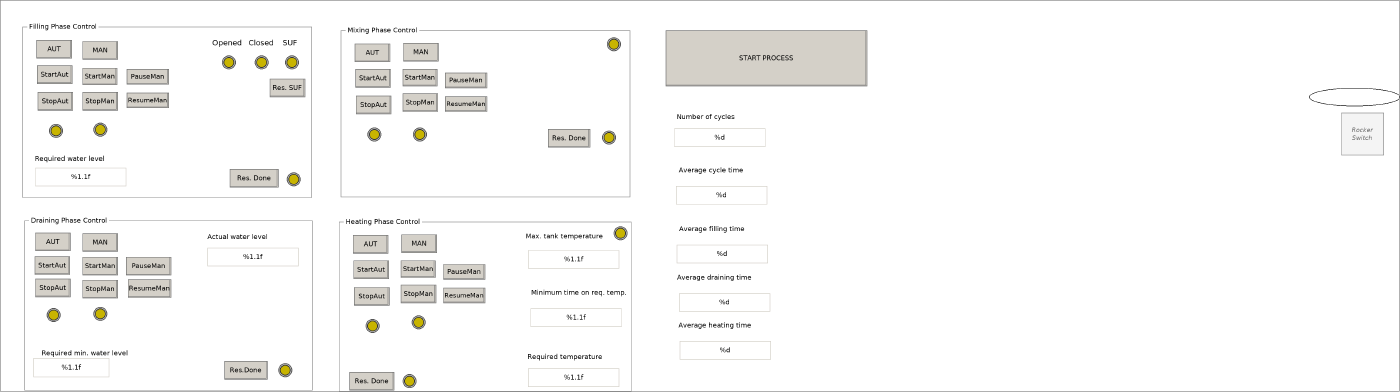
VISUALIZATION Visualization  // 2309x647
    GroupBox (40,356 475x288), "Draining Phase Control"
        Button (18,28 58x30), "AUT"
            OnMouseClick: toggle Global.Tank1.Draining.Cmd.AutCtrl
        Button (96,29 58x30), "MAN"
            OnMouseClick: toggle Global.Tank1.Draining.Cmd.ManCtrl
        Button (17,67 58x30), "StartAut"
            OnMouseClick: toggle Global.Tank1.Draining.Cmd.StartAut
        Button (168,68 74x30), "PauseMan"
            OnMouseClick: toggle Global.Tank1.Draining.Cmd.PauseMan
        Button (96,68 58x30), "StartMan"
            OnMouseClick: toggle Global.Tank1.Draining.Cmd.StartMan
        Button (96,106 58x30), "StopMan"
            OnMouseClick: toggle Global.Tank1.Draining.Cmd.StopMan
        Button (171,105 71x30), "ResumeMan"
            OnMouseClick: toggle Global.Tank1.Draining.Cmd.ResumeMan
        Button (18,104 58x30), "StopAut"
            OnMouseClick: toggle Global.Tank1.Draining.Cmd.StopAut
        Button (330,240 71x30), "Res.Done"
            OnMouseClick: toggle Global.Tank1.Draining.Cmd.ResetDone
        Lamp1 (417,242 27x26), variable: Global.Tank1.Draining.State.Done, style: Lamp-Lamp1-Yellow
        Lamp1 (35,151 27x26), variable: Global.Tank1.Draining.State.AutCtrl, style: Lamp-Lamp1-Yellow
        Lamp1 (112,149 27x26), variable: Global.Tank1.Draining.State.ManCtrl, style: Lamp-Lamp1-Yellow
        Textfield (302,53 150x30), "%1.1f", text variable: Global.Tank1.Draining.WaterLevel
        Textfield (15,235 125x31), "%1.1f", text variable: Global.Tank1.Draining.ParamDrainLevel
            OnMouseDown: write Global.Tank1.Draining.ParamDrainLevel via Edit
        Label (277,20 150x30), "Actual water level"
        Label (25,212 150x30), "Required min. water level"
    RockerSwitch (2212,186 70x70), behaviour: TOGGLE, style: Switch-RockerSwitch-Gray
    Ellipse (2159,145 150x30)
    GroupBox (37,36 477x290), "Filling Phase Control"
        Button (23,30 58x30), "AUT", text variable: Global.Tank1.Filling.Cmd.AutCtrl
            OnMouseClick: toggle Global.Tank1.Filling.Cmd.AutCtrl
        Button (99,32 58x30), "MAN"
            OnMouseClick: toggle Global.Tank1.Filling.Cmd.ManCtrl
        Button (24,72 58x30), "StartAut"
            OnMouseClick: toggle Global.Tank1.Filling.Cmd.StartAut
        Button (25,116 58x30), "StopAut"
            OnMouseClick: toggle Global.Tank1.Filling.Cmd.StopAut
        Button (342,243 80x30), "Res. Done"
            OnMouseClick: toggle Global.Tank1.Filling.Cmd.ResetDone
        Lamp1 (434,247 27x26), variable: Global.Tank1.Filling.State.Done, style: Lamp-Lamp1-Yellow
        Textfield (21,241 150x30), "%1.1f", text variable: Global.Tank1.Filling.ParamFillLevel
            OnMouseDown: write Global.Tank1.Filling.ParamFillLevel via Edit
        Button (99,76 57x28), "StartMan"
            OnMouseClick: toggle Global.Tank1.Filling.Cmd.StartMan
        Button (99,116 58x30), "StopMan"
            OnMouseClick: toggle Global.Tank1.Filling.Cmd.StopMan
        Lamp1 (115,165 27x26), variable: Global.Tank1.ValveFilling.State.ManCtrl, style: Lamp-Lamp1-Yellow
        Lamp1 (42,167 27x26), variable: Global.Tank1.ValveFilling.State.AutCtrl, style: Lamp-Lamp1-Yellow
        Button (172,78 69x25), "PauseMan"
            OnMouseDown: toggle Global.Tank1.Filling.Cmd.PauseMan
        Button (172,117 69x25), "ResumeMan"
            OnMouseDown: toggle Global.Tank1.Filling.Cmd.ResumeMan
        Button (408,94 58x30), "Res. SUF", text variable: Global.Tank1.ValveFilling.Cmd.ResetSUF
            OnMouseClick: toggle Global.Tank1.ValveFilling.Cmd.ResetSUF
        Lamp1 (431,54 27x26), variable: Global.Tank1.ValveFilling.State.StartupFail, style: Lamp-Lamp1-Yellow
        Lamp1 (327,54 27x26), variable: Global.Tank1.ValveFilling.State.Open, style: Lamp-Lamp1-Yellow
        Lamp1 (381,54 27x26), variable: Global.Tank1.ValveFilling.State.Closed, style: Lamp-Lamp1-Yellow
        Label (310,26 53x18), "Opened"
        Label (370,26 53x18), "Closed"
        Label (426,26 33x18), "SUF"
        Label (3,211 150x30), "Required water level"
    GroupBox (562,42 477x283), "Mixing Phase Control"
        Button (23,30 58x30), "AUT", text variable: Global.Tank1.Filling.Cmd.AutCtrl
            OnMouseClick: toggle Global.Tank1.Mixing.Cmd.AutCtrl
        Button (103,29 58x30), "MAN"
            OnMouseClick: toggle Global.Tank1.Mixing.Cmd.ManCtrl
        Button (24,72 58x30), "StartAut"
            OnMouseClick: toggle Global.Tank1.Mixing.Cmd.StartAut
        Button (25,116 58x30), "StopAut"
            OnMouseClick: toggle Global.Tank1.Mixing.Cmd.StopAut
        Button (342,171 69x30), "Res. Done"
            OnMouseClick: toggle Global.Tank1.Mixing.Cmd.ResetDone
        Lamp1 (429,172 27x26), variable: Global.Tank1.Mixing.State.Done, style: Lamp-Lamp1-Yellow
        Button (102,72 57x28), "StartMan"
            OnMouseClick: toggle Global.Tank1.Mixing.Cmd.StartMan
        Button (102,112 58x30), "StopMan"
            OnMouseClick: toggle Global.Tank1.Mixing.Cmd.StopMan
        Lamp1 (117,167 27x26), variable: Global.Tank1.Mixer.State.ManCtrl, style: Lamp-Lamp1-Yellow
        Lamp1 (42,167 27x26), variable: Global.Tank1.Mixer.State.AutCtrl, style: Lamp-Lamp1-Yellow
        Button (172,78 69x25), "PauseMan"
            OnMouseDown: toggle Global.Tank1.Mixing.Cmd.PauseMan
        Button (172,117 69x25), "ResumeMan"
            OnMouseDown: toggle Global.Tank1.Mixing.Cmd.ResumeMan
        Lamp1 (437,18 27x26), variable: Global.Tank1.Mixer.State.RunOut, style: Lamp-Lamp1-Yellow
    GroupBox (559,358 482x289), "Heating Phase Control"
        Button (23,30 58x30), "AUT", text variable: Global.Tank1.Filling.Cmd.AutCtrl
            OnMouseClick: toggle Global.Tank1.Heating.Cmd.AutCtrl
        Button (103,29 58x30), "MAN"
            OnMouseClick: toggle Global.Tank1.Heating.Cmd.ManCtrl
        Button (24,72 58x30), "StartAut"
            OnMouseClick: toggle Global.Tank1.Heating.Cmd.StartAut
        Button (25,116 58x30), "StopAut"
            OnMouseClick: toggle Global.Tank1.Heating.Cmd.StopAut
        Button (17,256 74x30), "Res. Done"
            OnMouseClick: toggle Global.Tank1.Heating.Cmd.ResetDone
        Lamp1 (103,258 27x26), variable: Global.Tank1.Heating.State.Done, style: Lamp-Lamp1-Yellow
        Button (102,72 57x28), "StartMan"
            OnMouseClick: toggle Global.Tank1.Heating.Cmd.StartMan
        Button (102,112 58x30), "StopMan"
            OnMouseClick: toggle Global.Tank1.Heating.Cmd.StopMan
        Lamp1 (118,161 27x26), variable: Global.Tank1.Heater.State.ManCtrl, style: Lamp-Lamp1-Yellow
        Lamp1 (42,167 27x26), variable: Global.Tank1.Heater.State.AutCtrl, style: Lamp-Lamp1-Yellow
        Button (172,78 69x25), "PauseMan"
            OnMouseDown: toggle Global.Tank1.Heating.Cmd.PauseMan
        Button (172,117 69x25), "ResumeMan"
            OnMouseDown: toggle Global.Tank1.Heating.Cmd.ResumeMan
        Textfield (312,250 150x30), "%1.1f", text variable: Global.Tank1.Heating.ParamReqTemp
            OnMouseDown: write Global.Tank1.Heating.ParamReqTemp via Edit
        Textfield (316,151 150x30), "%1.1f", text variable: Global.timeReqOnTemp
            OnMouseDown: write Global.timeReqOnTemp via Edit
        Textfield (312,55 150x30), "%1.1f", text variable: Global.maxWaterTemp
            OnMouseDown: write Global.maxWaterTemp via Edit
        Label (298,216 150x30), "Required temperature"
        Label (297,17 150x30), "Max. tank temperature"
        Label (315,110 162x30), "Minimum time on req. temp."
        Lamp1 (451,14 27x26), variable: Global.Tank1.Heater.State.EnableOut, style: Lamp-Lamp1-Yellow
    Button (1098,50 332x92), "START PROCESS"
        OnMouseClick: toggle MAIN.start_process
    Textfield (1115,307 150x30), "%d", text variable: Global.avgCycleTime
    Textfield (1112,212 150x30), "%d", text variable: Global.cycleCount
    Label (1098,266 150x30), "Average cycle time"
    Label (1089,178 150x30), "Number of cycles"
    Textfield (1116,404 150x30), "%d", text variable: Global.AvgFillingTime
    Label (1099,363 150x30), "Average filling time"
    Textfield (1121,563 150x30), "%d", text variable: Global.AvgHeatingTime
    Label (1104,522 150x30), "Average heating time"
    Textfield (1120,484 150x30), "%d", text variable: Global.AvgDrainingTime
    Label (1103,443 150x30), "Average draining time"
END_VISUALIZATION

(* stored: Version 1.1.0.1, ProductVersion 3.1.4024.13
   Visu Visualization: Id {a6343251-0068-49ba-9adb-31cb88a6e465} *)
